{attribute 'GeneratedUsingTerminal: EPP9022-0060-0017'}
{attribute addProperty BoxType "EPP9022-0060-0017"}
{attribute addProperty Id "EtcSlaveTerminalBaseEPM_Inputs_Channel_1AT %I*EPM_Inputs_Channel_B9246B8D18EPM_Inputs_Channel_2AT %I*EPM_Inputs_Channel_B9246B8D18WcStateAT %I*WcState_9091E0EB2InfoDataAT %I*InfoData_32EB74EA10"}
{attribute addProperty CRC "3727263012"}
{attribute addProperty Size "48"}
TYPE EPP9022_DE298524 EXTENDS EtcSlaveTerminalBase :
STRUCT
	{attribute addProperty Name "EPM_Inputs_Channel_1"}
	EPM_Inputs_Channel_1 : EPM_Inputs_Channel_B9246B8D;
	{attribute addProperty Name "EPM_Inputs_Channel_2"}
	EPM_Inputs_Channel_2 : EPM_Inputs_Channel_B9246B8D;
	{attribute addProperty Name "WcState"}
	WcState : WcState_9091E0EB;
	{attribute addProperty Name "InfoData"}
	InfoData : InfoData_32EB74EA;
END_STRUCT
END_TYPE

(* stored: Version 1.2.0.0, ProductVersion 3.1.4024.9
   DUT EPP9022_DE298524: Id {c0dd26b5-1924-43d4-b353-8e4c27bc2525} *)
